(* PLC project Programme MGS_2-07_refactorJOY.project, CODESYS CODESYS V3.5 SP19 Patch 1 *)
(* stored: creationDateTime 2026-06-29T23:37:40.2944815, modificationDateTime 2026-06-29T22:49:33.424 *)

FUNCTION_BLOCK FB_Filter_PT1
  VAR_INPUT
    ValueIn : REAL;  (* Consigne brute entrée *)
    TimeConst : TIME;  (* Constante de temps du filtre *)
    CycleTimeS : REAL;  (* Temps de cycle réel en secondes *)
    Enable : BOOL;  (* Active le filtre *)
  END_VAR
  VAR_OUTPUT
    ValueOut : REAL;  (* Consigne filtrée sortie *)
  END_VAR
  VAR
    T : REAL;
    Alpha : REAL;
  END_VAR

            T := TIME_TO_REAL(TimeConst) / 1000.0;

IF (T + CycleTimeS) > 0.0 THEN
    Alpha := CycleTimeS / (T + CycleTimeS);
    ValueOut := ValueOut + Alpha * (ValueIn - ValueOut);
ELSE
    ValueOut := ValueIn;
END_IF;
          
END_FUNCTION_BLOCK
